FUNCTION_BLOCK ProfibusDeviceBase
VAR_INPUT
END_VAR
VAR_OUTPUT
END_VAR
VAR
	DpState AT%I* : USINT;
	ExtDiagFlag at%i* : BOOL;
END_VAR

END_FUNCTION_BLOCK

(* stored: Version 1.1.0.1, ProductVersion 3.1.4024.11
   POU ProfibusDeviceBase: Id {47c4ad1f-9b3f-4c9b-9734-d4706eb3885a}, SpecialFunc None *)
